// TIA Portal V17 export
// export: Created 2022-07-20T07:02:39.3280098Z, ExportSetting WithDefaults, DisplayName Totally Integrated Automation Portal, DisplayVersion V17, DisplayName TIA Portal Openness, DisplayVersion V17, DisplayName TIA Portal Version Control Interface, DisplayVersion V17, DisplayName SINAMICS Startdrive Advanced, DisplayVersion V17, DisplayName SINAMICS Startdrive G130, G150, S120, S150, SINAMICS MV, S210, DisplayVersion V17, DisplayName SINAMICS Startdrive G110M, G120, G120C, G120D, G120P, G115D, DisplayVersion V17, DisplayName STEP 7 Professional, DisplayVersion V17, DisplayName STEP 7 Safety, DisplayVersion V17, DisplayName WinCC Advanced, DisplayVersion V17
VAR_GLOBAL   // PLC tag table "ELGuider_Webguide_CommunicationTable"
   Elguiderv2In_0 AT %IW916 : Int;
   Elguiderv2In_1 AT %IW918 : Int;
   Elguiderv2In_2 AT %IW920 : Int;
   Elguiderv2In_3 AT %IW922 : Int;
   Elguiderv2In_4 AT %IW924 : Int;
   Elguiderv2In_5 AT %IW926 : Int;
   Elguiderv2In_6 AT %IW928 : Int;
   Elguiderv2In_7 AT %IW930 : Int;
   Elguiderv2In_8 AT %IW932 : Int;
   Elguiderv2In_9 AT %IW934 : Int;
   Elguiderv2In_10 AT %IW936 : Int;
   Elguiderv2In_11 AT %IW938 : Int;
   Elguiderv2In_12 AT %IW940 : Int;
   Elguiderv2In_13 AT %IW942 : Int;
   Elguiderv2In_14 AT %IW944 : Int;
   Elguiderv2In_15 AT %IW946 : Int;
   Elguiderv2In_16 AT %IW948 : Int;
   Elguiderv2In_17 AT %IW950 : Int;
   Elguiderv2In_18 AT %IW952 : Int;
   Elguiderv2In_19 AT %IW954 : Int;
   Elguiderv2In_20 AT %IW956 : Int;
   Elguiderv2In_21 AT %IW958 : Int;
   Elguiderv2In_22 AT %IW960 : Int;
   Elguiderv2In_23 AT %IW962 : Int;
   Elguiderv2In_24 AT %IW964 : Int;
   Elguiderv2In_25 AT %IW966 : Int;
   Elguiderv2In_26 AT %IW968 : Int;
   Elguiderv2In_27 AT %IW970 : Int;
   Elguiderv2In_28 AT %IW972 : Int;
   Elguiderv2Out_0 AT %QW866 : Int;
   Elguiderv2Out_1 AT %QW868 : Int;
   Elguiderv2Out_2 AT %QW870 : Int;
   Elguiderv2Out_3 AT %QW872 : Int;
   Elguiderv2Out_4 AT %QW874 : Int;
   Elguiderv2Out_5 AT %QW876 : Int;
   Elguiderv2Out_6 AT %QW878 : Int;
   Elguiderv2Out_7 AT %QW880 : Int;
   Elguiderv2Out_8 AT %QW882 : Int;
   Elguiderv2Out_9 AT %QW884 : Int;
   Elguiderv2Out_10 AT %QW886 : Int;
   Elguiderv2Out_11 AT %QW888 : Int;
   Elguiderv2Out_12 AT %QW890 : Int;
   Elguiderv2Out_13 AT %QW892 : Int;
   Elguiderv2Out_14 AT %QW894 : Int;
   Elguiderv2Out_15 AT %QW896 : Int;
   Elguiderv2Out_16 AT %QW898 : Int;
   Elguiderv2Out_17 AT %QW900 : Int;
   Elguiderv2Out_18 AT %QW902 : Int;
   Elguiderv2Out_19 AT %QW904 : Int;
   Elguiderv2Out_20 AT %QW906 : Int;
   Elguiderv2Out_21 AT %QW908 : Int;
   Elguiderv2Out_22 AT %QW910 : Int;
   Elguiderv2Out_23 AT %QW912 : Int;
   Elguiderv2Out_24 AT %QW914 : Int;
   Elguiderv2Out_25 AT %QW916 : Int;
   Elguiderv2Out_26 AT %QW918 : Int;
   Elguiderv2Out_27 AT %QW920 : Int;
   Elguiderv2Out_28 AT %QW922 : Int;
END_VAR
